Staubli VAL3: ExampleTest.pgx

program ExampleTest()
  local num l_nStart
  local num l_nEnd
  local bool l_bRes
  local num l_nNum
  local string l_sBuff
begin


  //××××××××××××××××××××××××××××××××××××××××××××××××××××××××××××××××××××××××××××××××××××
  //××××××××××××××××××××××××××××××××××××××××××××××××××××××××××××××××××××××××××××××××××××
  //把product文件中的某条路径给替换掉
  //





  //查询
  call GetTrajFlag(l_bRes,"Disk://product1.txt",3,l_nStart,l_nEnd)
  if !l_bRes
    return
  endIf


  //产生文件
  call CreatFile("Disk://Buff.txt",l_bRes)
  if !l_bRes
    return
  endIf

  //添加开头
  call CopyFileContext(l_bRes,"Disk://product1.txt","Disk://Buff.txt",0,l_nStart-2)
  if !l_bRes
    return
  endIf
  //***************************************************************************************
  //输入内容
  nFileID=$fileOpen("Disk://Buff.txt","a")
  if nFileID<0 or nFileID>9
    return
  endIf

  l_sBuff="=BEGIN"
  l_nNum=$fileSet(nFileID,l_sBuff,l_nNum)

  for l_nNum=0 to 100
    l_sBuff=toString("",l_nNum)
    if $fileSet(nFileID,l_sBuff,1)!=1
      return
    endIf
  endFor

  l_sBuff="=END"
  l_nNum=$fileSet(nFileID,l_sBuff,l_nNum)
  call CloseAllFile()
  //************************************************************************************

  //把末尾给附加上去
  call CopyFileContext(l_bRes,"Disk://product1.txt","Disk://Buff.txt",l_nEnd+1,-1)
  if !l_bRes
    return
  endIf

  //把临时文件给删除掉
  //使用rename必须把需要命名的文件的名字不能存在，否则报错
  $delete("Disk://product1.txt")
  if !$rename("Disk://Buff.txt","Disk://product1.txt")
  endIf
end
